(* CODESYS project SumAndSubtract.project

Project tree, tasks and I/O mapping:
  Device : CODESYS Control Win V3, 3S - Smart Software Solutions GmbH, version 3.5.15.30
    application Application
      libraries: Standard, * (System)
      task MainTask (cyclic, interval t#20ms, priority 1) calls PLC_PRG, FBD_PRG
      program PLC_PRG [ST]
      function block SumAndSubtract_FB [ST]
      program FBD_PRG [FBD]
*)

// Device/Application/PLC_PRG
PROGRAM PLC_PRG
VAR
	A : REAL := 11;
	B : REAL := 5;
	Sum : REAL;
	Subtr : REAL;
	
	MyFB : SumAndSubtract_FB;
END_VAR

(* Invoke the FB explicitly binding params to PRG vars *)
MyFB(num1 := A, num2 := B);

(* Assign return values *)
Sum := MyFB.SumResult;
Subtr := MyFB.SubResult;

END_PROGRAM

// Device/Application/SumAndSubtract_FB
FUNCTION_BLOCK SumAndSubtract_FB

VAR_INPUT
	num1 : REAL;
	num2 : REAL;
END_VAR

VAR_OUTPUT
	SumResult : REAL;
	SubResult : REAL;
END_VAR

VAR
	(* No internal vars... *)
END_VAR

SumResult := num1 + num2;
SubResult := num1 - num2;

END_FUNCTION_BLOCK

// Device/Application/FBD_PRG
PROGRAM FBD_PRG
VAR
	A : REAL := 11;
	B : REAL := 5;
	Sum : REAL;
	Subtr : REAL;
	
	SumAndSubtract_FB_0: SumAndSubtract_FB;
END_VAR

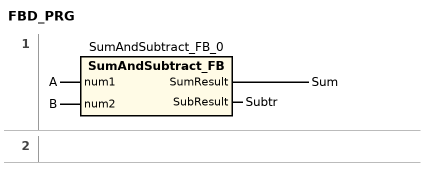
// NETWORK 1
SumAndSubtract_FB_0(num1 := A, num2 := B, SubResult => Subtr); // SumAndSubtract_FB
Sum := SumAndSubtract_FB_0.SumResult;

// NETWORK 2

END_PROGRAM
